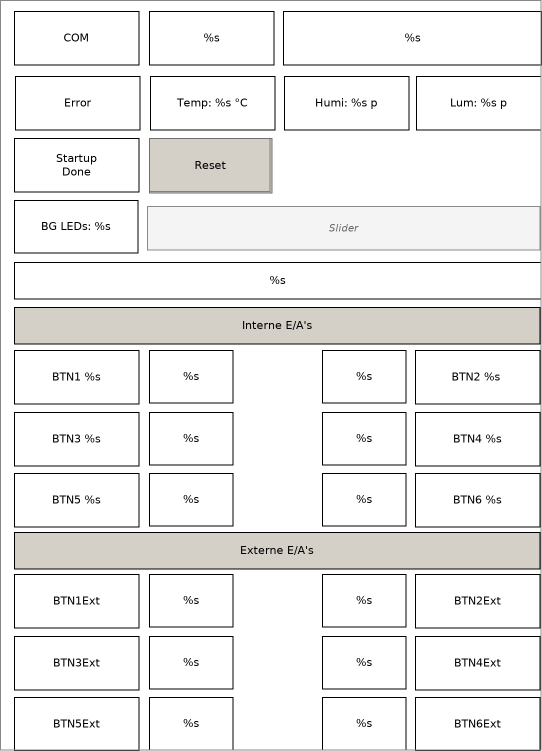
VISUALIZATION BusTatster6F_Frame_1  // 542x751
VAR_IN_OUT
	stBusTaster6F_Input		:ST_BusTaster6F_Input;
	stBusTaster6F_Output	:ST_BusTaster6F_Output;
	stBusTaster6F_Cnt		:ST_BusTaster6F_Cnt;
END_VAR
    Rectangle (14,11 125x54), "COM", colour toggle: stBusTaster6F_Output.bCOM
    Rectangle (14,350 125x54), "BTN1 %s", text variable: stBusTaster6F_Cnt.dwCntButtons[1], colour toggle: stBusTaster6F_Output.bButtons[1]
    Rectangle (149,11 125x54), "%s", text variable: stBusTaster6F_Input.diID
    Rectangle (283,11 259x54), "%s", text variable: stBusTaster6F_Input.sName
    Rectangle (415,350 125x54), "BTN2 %s", text variable: stBusTaster6F_Cnt.dwCntButtons[2], colour toggle: stBusTaster6F_Output.bButtons[2]
    Rectangle (14,412 125x54), "BTN3 %s", text variable: stBusTaster6F_Cnt.dwCntButtons[3], colour toggle: stBusTaster6F_Output.bButtons[3]
    Rectangle (415,412 125x54), "BTN4 %s", text variable: stBusTaster6F_Cnt.dwCntButtons[4], colour toggle: stBusTaster6F_Output.bButtons[4]
    Rectangle (14,473 125x54), "BTN5 %s", text variable: stBusTaster6F_Cnt.dwCntButtons[5], colour toggle: stBusTaster6F_Output.bButtons[5]
    Rectangle (415,473 125x54), "BTN6 %s", text variable: stBusTaster6F_Cnt.dwCntButtons[6], colour toggle: stBusTaster6F_Output.bButtons[6]
    Rectangle (149,350 84x53), "%s", text variable: stBusTaster6F_Input.iLED[1]
        OnMouseDown: write the text variable via VisuDialogs.Numpad, min 0, max 100
    Rectangle (322,350 84x53), "%s", text variable: stBusTaster6F_Input.iLED[2]
        OnMouseDown: write the text variable via VisuDialogs.Numpad, min 0, max 100
    Rectangle (149,412 84x53), "%s", text variable: stBusTaster6F_Input.iLED[3]
        OnMouseDown: write the text variable via VisuDialogs.Numpad, min 0, max 100
    Rectangle (322,412 84x53), "%s", text variable: stBusTaster6F_Input.iLED[4]
        OnMouseDown: write the text variable via VisuDialogs.Numpad, min 0, max 100
    Rectangle (149,473 84x53), "%s", text variable: stBusTaster6F_Input.iLED[5]
        OnMouseDown: write the text variable via VisuDialogs.Numpad, min 0, max 100
    Rectangle (322,473 84x53), "%s", text variable: stBusTaster6F_Input.iLED[6]
        OnMouseDown: write the text variable via VisuDialogs.Numpad, min 0, max 100
    Button (149,138 123x55), "Reset"
        tap stBusTaster6F_Input.bReset
    Rectangle (15,76 125x54), "Error", colour toggle: stBusTaster6F_Output.bError
    Rectangle (150,76 125x54), "Temp: %s °C", text variable: stBusTaster6F_Output.lrTemp
    Rectangle (284,76 125x54), "Humi: %s p", text variable: stBusTaster6F_Output.lrRhd
    Rectangle (416,76 125x54), "Lum: %s p", text variable: stBusTaster6F_Output.lrBrs
    Rectangle (14,262 527x37), "%s", text variable: stBusTaster6F_Output.sState
    Rectangle (14,138 125x54), "Startup Done", colour toggle: stBusTaster6F_Output.bStartupDone
    Rectangle (14,200 124x53), "BG LEDs: %s", text variable: stBusTaster6F_Input.iLEDBg
        OnMouseDown: write the text variable via VisuDialogs.Numpad, min 0, max 100
    Rectangle (14,574 125x54), "BTN1Ext", colour toggle: stBusTaster6F_Output.bButtonsExt[1]
    Rectangle (415,574 125x54), "BTN2Ext", colour toggle: stBusTaster6F_Output.bButtonsExt[2]
    Rectangle (14,636 125x54), "BTN3Ext", colour toggle: stBusTaster6F_Output.bButtonsExt[3]
    Rectangle (415,636 125x54), "BTN4Ext", colour toggle: stBusTaster6F_Output.bButtonsExt[4]
    Rectangle (14,697 125x54), "BTN5Ext", colour toggle: stBusTaster6F_Output.bButtonsExt[5]
    Rectangle (415,697 125x54), "BTN6Ext", colour toggle: stBusTaster6F_Output.bButtonsExt[6]
    Rectangle (149,574 84x53), "%s", text variable: stBusTaster6F_Input.iLEDExt[1]
        OnMouseDown: write the text variable via VisuDialogs.Numpad, min 0, max 100
    Rectangle (322,574 84x53), "%s", text variable: stBusTaster6F_Input.iLEDExt[2]
        OnMouseDown: write the text variable via VisuDialogs.Numpad, min 0, max 100
    Rectangle (149,636 84x53), "%s", text variable: stBusTaster6F_Input.iLEDExt[3]
        OnMouseDown: write the text variable via VisuDialogs.Numpad, min 0, max 100
    Rectangle (322,636 84x53), "%s", text variable: stBusTaster6F_Input.iLEDExt[4]
        OnMouseDown: write the text variable via VisuDialogs.Numpad, min 0, max 100
    Rectangle (149,697 84x53), "%s", text variable: stBusTaster6F_Input.iLEDExt[5]
        OnMouseDown: write the text variable via VisuDialogs.Numpad, min 0, max 100
    Rectangle (322,697 84x53), "%s", text variable: stBusTaster6F_Input.iLEDExt[6]
        OnMouseDown: write the text variable via VisuDialogs.Numpad, min 0, max 100
    Rectangle (14,532 526x37), "Externe E/A's"
    Rectangle (14,307 526x37), "Interne E/A's"
    Slider (147,206 393x44), variable: stBusTaster6F_Input.iLEDBg, scale 0..100
END_VISUALIZATION

(* stored: Version 1.1.0.1, ProductVersion 3.1.4024.12
   Visu BusTatster6F_Frame_1: Id {1f15b8af-12fd-4b09-8208-6db846e5398f} *)
